KUKA KRL program: style_1.src, style_1.dat

--- style_1.src ---
&ACCESS RVO1
&REL 101
&COMMENT 03-10-R1 STYLE 1
DEF Style_1( )
   ;FOLD INI;%{PE}
      ;FOLD BASISTECH INI
         GLOBAL INTERRUPT DECL 3 WHEN $STOPMESS==TRUE DO IR_STOPM ( )
         INTERRUPT ON 3
         BAS (#INITMOV,0 )
      ;ENDFOLD (BASISTECH INI)
      ;FOLD USER INI
         ;Make your modifications here

      ;ENDFOLD (USER INI)
   ;ENDFOLD (INI)
;********************************
; Gestamp Standards
; Line - BMW G65 (cell 03)
; Robot 03-10-R1 (BMW-03-10-R1)
; Application - STYLE 1: SELECT THE OPTION PROGRAM
;********************************
   ;SELECT THE OPTION PROGRAM BY OPTION NUMBER nOption (gdiOption $IN[38..45])
   SWITCH nOption
      CASE 1
         ;OPTION 1: PRODUCTION CYCLE (PICK, WELD 3 NUTS, NUT CHECKS, DROP OR REJECT)
         Style1Opt1 ( )
      CASE 2
         ;OPTION 2: SAME PRODUCTION CYCLE (Style1Opt1)
         ;NOTE: THE NUT SENSOR CHECK EVALUATES ONLY OPTIONS 1 AND 10 - FOR OPTIONS 2/7/8 ONLY THE
         ;NOTE: CAMERA DECIDES SCRAP OR GOOD (F02)
         Style1Opt1 ( )
      CASE 7
         ;OPTION 7: SAME PRODUCTION CYCLE (Style1Opt1) - NUT SENSOR NOT EVALUATED (F02)
         Style1Opt1 ( )
      CASE 8
         ;OPTION 8: SAME PRODUCTION CYCLE (Style1Opt1) - NUT SENSOR NOT EVALUATED (F02)
         Style1Opt1 ( )
      CASE 12
         ;OPTION 12: RED RABBIT TEST CYCLE (Style1Opt10AutoRR)
         ;NOTE: THE NUT CHECK EVALUATES THE RED RABBIT ONLY FOR OPTION 10, NOT 12 (F19)
         Style1Opt10AutoRR ( )
      DEFAULT
         ;NOTE: ANY OTHER OPTION: WAIT FOR FALSE - THE ROBOT STOPS HERE IN CYCLE FOR EVER,
         ;NOTE: WITH NO MESSAGE AND NO FAULT TO THE PLC (F06, C21)
         WAIT FOR FALSE
   ENDSWITCH



END

--- style_1.dat ---
&ACCESS RVO1
&REL 101
&COMMENT GE4_002
DEFDAT  style_1
;FOLD EXTERNAL DECLARATIONS;%{PE}%MKUKATPBASIS,%CEXT,%VCOMMON,%P
;FOLD BASISTECH EXT;%{PE}%MKUKATPBASIS,%CEXT,%VEXT,%P
EXT  BAS (BAS_COMMAND  :IN,REAL  :IN )
DECL INT SUCCESS
;ENDFOLD (BASISTECH EXT)
;FOLD USER EXT;%{E}%MKUKATPUSER,%CEXT,%VEXT,%P
;Make your modifications here

;ENDFOLD (USER EXT)
;ENDFOLD (EXTERNAL DECLARATIONS)
DECL BASIS_SUGG_T LAST_BASIS={POINT1[] "POUNCE                  ",POINT2[] "POUNCE                  ",CP_PARAMS[] "CPDAT0                  ",PTP_PARAMS[] "PDAT6                   ",CONT[] "                        ",CP_VEL[] "2.0                     ",PTP_VEL[] "90                      ",SYNC_PARAMS[] "SYNCDAT                 ",SPL_NAME[] "S0                      ",A_PARAMS[] "ADAT0                   "}
ENDDAT
